(* IEC 61131-3 sources: brOscatLib/oscatNetw (part 4) *)

(* ---- MB_CLIENT.st ---- *)
FUNCTION_BLOCK MB_CLIENT
    (*http://www.oscat.de/images/OSCATBasic/oscat_basic333_en.pdf#page=112*)
    CASE state OF

    00: (* Warten auf DELAY-Time *)
    	ton_1(IN:=ENABLE,PT:=DELAY);

    	IF ton_1.Q OR DELAY = T#0s THEN
    		ton_1(IN:=FALSE);
    		state := 20;
    		ip_state := BYTE#1; (* Anmelden *)
    	END_IF

    20: (* Bei IP_Control anmelden *)
    	IF ip_state = BYTE#3 THEN
    		(* IP Datenverkehr einrichten *)
    		IP_C.C_PORT := WORD#0; (* Port von IP_CONTROL verwenden *)
    		IP_C.C_IP := DWORD#0; (* IP von IP_CONTROL verwenden *)
    		IP_C.C_MODE := BOOL_TO_BYTE(UDP); (* Mode: 0=TCP+ACTIVE+IP , 1=UDP+ACTIVE+IP *)
    		IP_C.TIME_RESET := TRUE; (* Zeitueberwachung rücksetzen *)
    		IP_C.C_ENABLE := TRUE; (* Verbindungsaufbau freigeben *)
    		IP_C.R_OBSERVE := TRUE; (* Empfangsueberwachung *)
    		ERROR := DWORD#00; (* letzten Fehler rücksetzen *)

    		CASE FC OF
    		(******************************************************************)
    		1..2: (* 0x01 Read Coil Status , 0x02 Read Input Status *)
    			IF R_POINTS <= 2000 THEN
    				w_tmp := INT_TO_WORD(R_ADDR);
    				S_BUF.BUFFER[08] := WORD_TO_BYTE(SHR(w_tmp,8));
    				S_BUF.BUFFER[09] := WORD_TO_BYTE(w_tmp);
    				w_tmp := INT_TO_WORD(R_POINTS);
    				S_BUF.BUFFER[10] := WORD_TO_BYTE(SHR(w_tmp,8));
    				S_BUF.BUFFER[11] := WORD_TO_BYTE(w_tmp);
    				S_BUF.SIZE := UINT#12;
    				response :=	WORD_TO_INT(SHR(INT_TO_WORD(R_POINTS + 7),3));
    				comp := 7;
    			ELSE
    				ERROR := DWORD#2; (* ILLEGAL DATA ADDRESS *)
    			END_IF
    		(******************************************************************)
    		3..4: (* 0x03 Read Holding Registers , 0x04 Read Input Registers *)
    			IF R_POINTS <= 125 THEN
    				w_tmp := INT_TO_WORD(R_ADDR);
    				S_BUF.BUFFER[08] := WORD_TO_BYTE(SHR(w_tmp,8));
    				S_BUF.BUFFER[09] := WORD_TO_BYTE(w_tmp);
    				w_tmp := INT_TO_WORD(R_POINTS);
    				S_BUF.BUFFER[10] := WORD_TO_BYTE(SHR(w_tmp,8));
    				S_BUF.BUFFER[11] := WORD_TO_BYTE(w_tmp);
    				S_BUF.SIZE := UINT#12;
    				response :=	WORD_TO_INT(SHL(w_tmp,1));
    				comp := 7;
    			ELSE
    				ERROR := DWORD#2; (* ILLEGAL DATA ADDRESS *)
    			END_IF
    		(******************************************************************)
    		5:	(* 0x05 Force Single Coil *)
    			IF W_DATA_ADR <= DATA_SIZE THEN
    				w_tmp := INT_TO_WORD(W_ADDR);
    				S_BUF.BUFFER[08] := WORD_TO_BYTE(SHR(w_tmp,8));
    				S_BUF.BUFFER[09] := WORD_TO_BYTE(w_tmp);
    				S_BUF.BUFFER[10] := SEL((DATA[W_DATA_ADR] AND SHL(WORD#1,W_DATA_BITPOS))>WORD#00,BYTE#16#00,BYTE#16#FF);
    				S_BUF.BUFFER[11] := BYTE#00;
    				S_BUF.SIZE := UINT#12;
    				response := 3;
    				comp := 11;
    			ELSE
    				ERROR := DWORD#2; (* ILLEGAL DATA ADDRESS *)
    			END_IF
    		(******************************************************************)
    		6:	(* 0x06 Preset Single Register *)
    			IF W_DATA_ADR <= DATA_SIZE THEN
    				w_tmp := INT_TO_WORD(W_ADDR);
    				S_BUF.BUFFER[08] := WORD_TO_BYTE(SHR(w_tmp,8));
    				S_BUF.BUFFER[09] := WORD_TO_BYTE(w_tmp);
    				w_tmp := DATA[W_DATA_ADR];
    				S_BUF.BUFFER[10] := WORD_TO_BYTE(SHR(w_tmp,8));
    				S_BUF.BUFFER[11] := WORD_TO_BYTE(w_tmp);
    				S_BUF.SIZE := UINT#12;
    				response := 3;
    				comp := 11;
    			ELSE
    				ERROR := DWORD#2; (* ILLEGAL DATA ADDRESS *)
    			END_IF
    		(******************************************************************)
    		15:	(* 0x0F Force Multiple Coils *)
    			IF (WORD_TO_INT(SHR(INT_TO_WORD(WORD_TO_INT(SHL(INT_TO_WORD(W_DATA_ADR),4)) + W_POINTS + W_DATA_BITPOS + 15),4)) <= DATA_SIZE) AND W_POINTS <= 1968 THEN
    				w_tmp := INT_TO_WORD(W_ADDR);
    				S_BUF.BUFFER[08] := WORD_TO_BYTE(SHR(w_tmp,8));
    				S_BUF.BUFFER[09] := WORD_TO_BYTE(w_tmp);
    				w_tmp := INT_TO_WORD(W_POINTS);
    				S_BUF.BUFFER[10] := WORD_TO_BYTE(SHR(w_tmp,8));
    				S_BUF.BUFFER[11] := WORD_TO_BYTE(w_tmp);
    				S_BUF.BUFFER[12] := WORD_TO_BYTE(SHR(INT_TO_WORD(W_POINTS + 7),3));

    				w_mask := SHL(WORD#1,W_DATA_BITPOS);
    				bit_pos := 0;
    				w_tmp := WORD#00;
    				idx1 := 12;
    				idx2 := W_DATA_ADR;
    				FOR i := 1 TO W_POINTS DO
    					w_tmp :=BIT_LOAD_W(w_tmp,(DATA[idx2] AND w_mask) > WORD#0,bit_pos);
    					bit_pos := bit_pos + 1;
    					IF bit_pos > 7 OR i=W_POINTS THEN
    						bit_pos := 0;
    						idx1 := idx1 + 1;
    						S_BUF.BUFFER[idx1] := WORD_TO_BYTE(w_tmp);
    						w_tmp := WORD#0;
    					END_IF
    					w_mask := ROL(w_mask,1);
    					IF w_mask = WORD#1 THEN
    						idx2 := idx2 +1;
    					END_IF
    				END_FOR
    				S_BUF.SIZE := INT_TO_UINT(idx1 + 1);
    				response := 3;
    				comp := 11;
    			ELSE
    				ERROR := DWORD#2; (* ILLEGAL DATA ADDRESS *)
    			END_IF
    		(******************************************************************)
    		16:	(* 0x10 Write Multiple Registers *)
    			IF W_DATA_ADR + W_POINTS <= DATA_SIZE AND W_POINTS <= 123 THEN
    				w_tmp := INT_TO_WORD(W_ADDR);
    				S_BUF.BUFFER[08] := WORD_TO_BYTE(SHR(w_tmp,8));
    				S_BUF.BUFFER[09] := WORD_TO_BYTE(w_tmp);
    				w_tmp := INT_TO_WORD(W_POINTS);
    				S_BUF.BUFFER[10] := WORD_TO_BYTE(SHR(w_tmp,8));
    				S_BUF.BUFFER[11] := WORD_TO_BYTE(w_tmp);
    				S_BUF.BUFFER[12] := SHL(S_BUF.BUFFER[11],1);

    				idx1 := 11;
    				count := W_DATA_ADR + W_POINTS - 1;
    				FOR i := W_DATA_ADR TO count DO
    					idx1 := idx1 + 2;
    					idx2 := idx1 + 1; (* zweiter index für pcworx notwendig ! *)
    					w_tmp := DATA[i];
    					S_BUF.BUFFER[idx1] := WORD_TO_BYTE(SHR(w_tmp,8));
    					S_BUF.BUFFER[idx2] := WORD_TO_BYTE(w_tmp);
    				END_FOR

    				S_BUF.SIZE := INT_TO_UINT(idx2 + 1);
    				response := 3;
    				comp := 11;
    			ELSE
    				ERROR := DWORD#2; (* ILLEGAL DATA ADDRESS *)
    			END_IF
    		(******************************************************************)
    		22:	(* 0x16 mask Write Register *)
    			IF W_DATA_ADR + 2 <= DATA_SIZE THEN
    				w_tmp := INT_TO_WORD(W_ADDR);
    				S_BUF.BUFFER[08] := WORD_TO_BYTE(SHR(w_tmp,8));
    				S_BUF.BUFFER[09] := WORD_TO_BYTE(w_tmp);
    				idx1 := W_DATA_ADR;
    				w_tmp := DATA[idx1];
    				S_BUF.BUFFER[10] := WORD_TO_BYTE(SHR(w_tmp,8));
    				S_BUF.BUFFER[11] := WORD_TO_BYTE(w_tmp);
    				idx1 := idx1 +1;
    				w_tmp := DATA[idx1];
    				S_BUF.BUFFER[12] := WORD_TO_BYTE(SHR(w_tmp,8));
    				S_BUF.BUFFER[13] := WORD_TO_BYTE(w_tmp);

    				S_BUF.SIZE := UINT#14;
    				response := 5;
    				comp := 13;
    			ELSE
    				ERROR := DWORD#2; (* ILLEGAL DATA ADDRESS *)
    			END_IF
    		(******************************************************************)
    		23:	(* 0x17 Read/Write Multible Registers *)
    			IF W_DATA_ADR + W_POINTS <= DATA_SIZE AND W_POINTS <= 121 AND R_POINTS <= 125 THEN
    				idx1 := 15;
    				count := W_DATA_ADR + W_POINTS - 1;
    				FOR i := W_DATA_ADR TO count DO
    					idx1 := idx1 + 2;
    					idx2 := idx1 + 1; (* zweiter index für pcworx notwendig ! *)
    					w_tmp := DATA[i];
    					S_BUF.BUFFER[idx1] := WORD_TO_BYTE(SHR(w_tmp,8));
    					S_BUF.BUFFER[idx2] := WORD_TO_BYTE(w_tmp);
    				END_FOR

    				(* WRITE *)
    				w_tmp := INT_TO_WORD(W_ADDR);
    				S_BUF.BUFFER[12] := WORD_TO_BYTE(SHR(w_tmp,8));
    				S_BUF.BUFFER[13] := WORD_TO_BYTE(w_tmp);
    				w_tmp := INT_TO_WORD(W_POINTS);
    				S_BUF.BUFFER[14] := WORD_TO_BYTE(SHR(w_tmp,8));
    				S_BUF.BUFFER[15] := WORD_TO_BYTE(w_tmp);
    				S_BUF.BUFFER[16] := SHL(S_BUF.BUFFER[15],1);

    				(* READ *)
    				w_tmp := INT_TO_WORD(R_ADDR);
    				S_BUF.BUFFER[08] := WORD_TO_BYTE(SHR(w_tmp,8));
    				S_BUF.BUFFER[09] := WORD_TO_BYTE(w_tmp);
    				w_tmp := INT_TO_WORD(R_POINTS);
    				S_BUF.BUFFER[10] := WORD_TO_BYTE(SHR(w_tmp,8));
    				S_BUF.BUFFER[11] := WORD_TO_BYTE(w_tmp);

    				S_BUF.SIZE := INT_TO_UINT(idx2 + 1);
    				response := WORD_TO_INT(SHL(w_tmp,1));
    				comp := 7;
    			ELSE
    				ERROR := DWORD#2; (* ILLEGAL DATA ADDRESS *)
    			END_IF
    		(******************************************************************)

    		ELSE
    			ERROR := DWORD#00000001; (* ILLEGAL FUNCTION *)
    		END_CASE

    		(* Daten senden *)
    		IF ERROR = DWORD#00 THEN
    			transaction_id := transaction_id + 1;
    			w_tmp := UINT_TO_WORD(S_BUF.SIZE - UINT#6);
    			(* ---- H E A D E R --------------------------------------------------------------- *)
    			S_BUF.BUFFER[0] := ip_id; (* TRANSACTION-ID HI-Byte *)
    			S_BUF.BUFFER[1] := INT_TO_BYTE(transaction_id); (* TRANSACTION-ID LO-Byte *)
    			S_BUF.BUFFER[2] := BYTE#00; (* PROTOKOLL-ID HI-Byte *)
    			S_BUF.BUFFER[3] := BYTE#00; (* PROTOKOLL-ID LO-Byte *)
    			S_BUF.BUFFER[4] := WORD_TO_BYTE(SHR(w_tmp,8)); (* Laenge HI-Byte *)
    			S_BUF.BUFFER[5] := WORD_TO_BYTE(w_tmp); (* Laenge LO-Byte *)
    			S_BUF.BUFFER[6] := UNIT_ID; (* UNIT *)
    			S_BUF.BUFFER[7] := INT_TO_BYTE(FC); (* FUNCTION-CODE *)
    			(*----- END OF HEADER --------------------------------------------------------------*)
    			R_BUF.SIZE := UINT#0; (* Empfangsbuffer löschen *)
    			state := 30; (* wait for response *)
    		ELSE
    			ip_state := BYTE#4; (* Abmelden *)
    			state := 00;
    		END_IF
    	END_IF

    30: (* response *)
    	IF IP_C.ERROR <> DWORD#00 THEN
    		ERROR := IP_C.ERROR;
    		ip_state := BYTE#4; (* Abmelden *)
    		state := 00;
    	ELSIF S_BUF.SIZE = UINT#0 AND R_BUF.SIZE > UINT#0 THEN
    		(* erwartete länge in sendebuffer nachträglich eintragen um vergleich zu ermöglichen *)
    		w_tmp := INT_TO_WORD(response + 3);
    		S_BUF.BUFFER[4] := WORD_TO_BYTE(SHR(w_tmp,8));
    		S_BUF.BUFFER[5] := WORD_TO_BYTE(w_tmp);

    		FOR i := 0 TO comp DO
    			IF S_BUF.BUFFER[i] <> R_BUF.BUFFER[i] THEN EXIT; END_IF
    		END_FOR

    		IF R_BUF.SIZE >= UINT#9 AND R_BUF.BUFFER[7] > BYTE#128 THEN  (* Bit 7 = ERROR Message *)
    			ERROR := BYTE_TO_DWORD(R_BUF.BUFFER[8]);
    			ip_state := BYTE#4; (* Abmelden *)
    			state := 00;
    		ELSIF R_BUF.SIZE = INT_TO_UINT(response + 9) AND i > comp THEN
    			mask := SHL(DWORD#1,FC);
    			(* READ_COILS, READ_INPUT_DISCRETES *)
    			IF (mask AND DWORD#2#00000000_00000000_00000000_00000110) > DWORD#0 THEN (* FC 1,2 *)
    				IF WORD_TO_INT(SHR(INT_TO_WORD(WORD_TO_INT(SHL(INT_TO_WORD(R_DATA_ADR),4)) + R_POINTS + R_DATA_BITPOS + 15),4)) <= DATA_SIZE THEN
    					b_mask := BYTE#1;
    					idx1 := 09;
    					idx2 := R_DATA_ADR;
    					bit_pos := R_DATA_BITPOS;
    					FOR i := 1 TO R_POINTS DO
    						DATA[idx2]:=BIT_LOAD_W(DATA[idx2],(R_BUF.BUFFER[idx1] AND b_mask) > BYTE#0,bit_pos);
    						bit_pos := bit_pos + 1;
    						IF bit_pos > 15 THEN
    							idx2 := idx2 + 1;
    							bit_pos := 0;
    						END_IF
    						b_mask := ROL(b_mask,1);
    						IF b_mask = BYTE#1 THEN
    							idx1 := idx1 + 1;
    						END_IF
    					END_FOR
    				ELSE
    					ERROR := DWORD#2; (* ILLEGAL DATA ADDRESS *)
    				END_IF

    			(* READ_MULTIPLE_REGISTERS, READ_INPUT_REGISTERS, READ_WRITE_REGISTERS *)
    			ELSIF (mask AND DWORD#2#00000000_10000000_00000000_00011000) > DWORD#0 THEN (* FC 3,4,23 *)
    				IF R_DATA_ADR + R_POINTS <= DATA_SIZE THEN
    					stop := R_DATA_ADR + R_POINTS -1 ;
    					idx1 := 07;
    					FOR i := R_DATA_ADR TO stop DO
    						idx1 := idx1 + 2;
    						idx2 := idx1 + 1;
    						DATA[i] := WORD_OF_BYTE(R_BUF.BUFFER[idx1],R_BUF.BUFFER[idx2]);
    					END_FOR
    				ELSE
    					ERROR := DWORD#2; (* ILLEGAL DATA ADDRESS *)
    				END_IF
    			ELSIF (mask AND DWORD#2#11111111_00111110_01111111_10000001) > DWORD#0 THEN (* ILLEGAL FUNCTION CODE ? *)
    				ERROR := DWORD#1; (* ILLEGAL FUNCTION *)
    			END_IF
    		ELSE
    			ERROR := DWORD#3; (* ILLEGAL DATA VALUE *)
    		END_IF

    		ip_state := BYTE#4; (* Abmelden *)
    		state := 00;
    		R_BUF.SIZE := UINT#0;

    	END_IF

    END_CASE

    (* ip_fifo *)
    ip_fifo(FIFO:=IP_C.FIFO,state:=ip_state,ID:=ip_id);
    BUSY := ip_state = BYTE#3;

    (* revision history
    ks	05. jan. 2009	rev 1.0
    	original version

    ks	28. jan. 2009	rev 1.1
    	network_buffer_short verwendet

    ks	20. oct. 2009	rev 1.2
    Networkbuffer und Buffer-funktionen auf Basis 0

    *)
END_FUNCTION_BLOCK

(* ---- MB_SERVER.st ---- *)
FUNCTION_BLOCK MB_SERVER
    (*http://www.oscat.de/images/OSCATBasic/oscat_basic333_en.pdf#page=116*)
    (* read system time *)
    tx := DWORD_TO_TIME(T_PLC_MS());

    FOR i := 1 TO 10 DO
    	IF VMAP[i].TIME_OUT > t#0s THEN
    		VMAP[i].TIME_OUT := VMAP[i].TIME_OUT + tx - last_cycle;
    	END_IF
    END_FOR
    last_cycle := tx;
    ip_error := IP_C.ERROR > DWORD#0;

    CASE state OF
    00: (* Warten auf Freigabe *)
    	IF ENABLE THEN
    		state := 10;
    		ip_state := BYTE#1; (* Anmelden *)
    	END_IF

    10: (* Bei IP_Control anmelden und auf freigabe warten *)
    	IF ip_state = BYTE#3 THEN

    		(* IP Datenverkehr einrichten *)
    		IP_C.C_PORT := WORD#0; (* Port von IP_CONTROL verwenden *)
    		IP_C.C_IP := DWORD#0; (* IP von IP_CONTROL verwenden *)
    		IP_C.C_MODE := SEL(UDP,BYTE#4,BYTE#5); (* Mode: 4=TCP+PASSIV+PORT , 5=UDP+PASSIV+PORT *)
    		IP_C.TIME_RESET := TRUE; (* Zeitueberwachung rücksetzen *)
    		IP_C.C_ENABLE := TRUE; (* Verbindungsaufbau freigeben *)
    		IP_C.R_OBSERVE := TRUE; (* keine Empfangsueberwachung *)
    		state := 20;
    	END_IF

    20:	IF NOT ip_error THEN
    		IF S_BUF.SIZE = UINT#0 AND R_BUF.SIZE > UINT#6 THEN	(* Datensenden nicht aktiv und Daten wurden empfangen *)
    			IF  R_BUF.SIZE = WORD_TO_UINT(WORD_OF_BYTE(R_BUF.BUFFER[4],R_BUF.BUFFER[5])) + UINT#6 THEN (* gültige Datenlänge *)
    				ERROR := DWORD#00; (* ERROR löschen *)

    				(* Header kopieren *)
    				FOR i := 0 TO 13 DO
    					S_BUF.BUFFER[i] := R_BUF.BUFFER[i];
    				END_FOR
    				fc := BYTE_TO_INT(R_BUF.BUFFER[7]);
    				adr1 := WORD_TO_INT(WORD_OF_BYTE(R_BUF.BUFFER[8],R_BUF.BUFFER[9]));
    				points := WORD_TO_INT(WORD_OF_BYTE(R_BUF.BUFFER[10],R_BUF.BUFFER[11]));

    				(* Virtual Address *)
    				MB_VMAP(VMAP:=VMAP,fc:=fc,V_ADR:=adr1,V_CNT:=points,SIZE:=DATA_SIZE);
    				adr1:=MB_VMAP.P_ADR;
    				bit_pos:=MB_VMAP.P_BIT;
    				ERROR:=BYTE_TO_DWORD(MB_VMAP.ERROR);

    				IF ERROR = DWORD#0 THEN
    					CASE fc OF
    					(*---------------------------------------------*)
    					1..2 : (* Read Coil Status / Read Input Status *)
    						count := 9; (* erstes Datenbyte *)
    						coils := BYTE#0;
    						mask := BYTE#1;
    						FOR i := 1 TO points DO
    							IF mask = BYTE#0 THEN
    								mask := BYTE#1;
    								S_BUF.BUFFER[count] := coils;
    								coils := BYTE#0;
    								count := count + 1;
    							END_IF
    							IF (DATA[adr1] AND SHL(WORD#1,bit_pos)) > WORD#0 THEN
    								coils := coils OR mask;
    							END_IF

    							bit_pos := bit_pos + 1;
    							IF bit_pos > 15 THEN
    								adr1 := adr1 + 1;
    								bit_pos := 0;
    							END_IF

    							mask := SHL(mask,1);
    						END_FOR
    						S_BUF.BUFFER[count] := coils;

    						S_BUF.BUFFER[8] := INT_TO_BYTE(count - 8); (* Bytecount *)
    						S_BUF.SIZE := INT_TO_UINT(count + 1);

    					(*--------------------------------------------------*)
    					3..4 : (* Read Holding Registers / Read Input Registers *)
    						idx1 := 07;
    						count := adr1 + points - 1;
    						FOR i := adr1 TO count DO
    							idx1 := idx1 + 2;
    							idx2 := idx1 + 1; (* zweiter index für pcworx notwendig ! *)
    							w_tmp := DATA[i];
    							S_BUF.BUFFER[idx1] := WORD_TO_BYTE(SHR(w_tmp,8));
    							S_BUF.BUFFER[idx2] := WORD_TO_BYTE(w_tmp);
    						END_FOR
    						S_BUF.BUFFER[8] := SHL(INT_TO_BYTE(points),1); (* Anzahl Register in Bytes *)
    						S_BUF.SIZE := INT_TO_UINT(idx2 + 1);
    					(*--------------------------------------------------*)
    					5 : (* Force Single Coil *)
    						DATA[adr1]:=BIT_LOAD_W(DATA[adr1],R_BUF.BUFFER[10] > BYTE#0,bit_pos);
    						S_BUF.SIZE := UINT#12;
    					(*--------------------------------------------------*)
    					6 : (* Preset Single Register *)
    						DATA[adr1] := WORD_OF_BYTE(R_BUF.BUFFER[10],R_BUF.BUFFER[11]);
    						S_BUF.SIZE := UINT#12;
    					(*--------------------------------------------------*)
    					15 : (* Force Multible coils *)
    						mask := BYTE#1;
    						idx1 := 13;
    						FOR i := 1 TO points DO
    							DATA[adr1]:=BIT_LOAD_W(DATA[adr1],(R_BUF.BUFFER[idx1] AND mask) > BYTE#0,bit_pos);
    							bit_pos := bit_pos + 1;
    							IF bit_pos > 15 THEN
    								adr1:= adr1 + 1;
    								bit_pos := 0;
    							END_IF
    							mask := ROL(mask,1);
    							IF mask = BYTE#1 THEN
    								idx1 := idx1 +1;
    							END_IF
    						END_FOR
    						S_BUF.SIZE := UINT#12;
    					(*--------------------------------------------------*)
    					16 : (* Preset Multiple Registers	*)
    						idx1 := 11;
    						count := adr1 + points - 1;
    						FOR i := adr1 TO count DO
    							idx1 := idx1 + 2;
    	 						idx2 := idx1 + 1;
    							DATA[i] := WORD_OF_BYTE(R_BUF.BUFFER[idx1],R_BUF.BUFFER[idx2]);
    						END_FOR
    						S_BUF.SIZE := UINT#12;
    					(*--------------------------------------------------*)
    					22 : (* mask Write Register *)
    						w_tmp := WORD_OF_BYTE(R_BUF.BUFFER[10],R_BUF.BUFFER[11]); (* and mask *)
    						DATA[adr1] := (DATA[adr1] AND w_tmp) OR (WORD_OF_BYTE(R_BUF.BUFFER[12],R_BUF.BUFFER[13]) AND (NOT w_tmp));
    						S_BUF.SIZE := UINT#14;
    					(*--------------------------------------------------*)
    					23 : (* Read / Write Registers	*)
    						(*--- Write-Register -----------------------------------*)
    						adr2 := WORD_TO_INT(WORD_OF_BYTE(R_BUF.BUFFER[12],R_BUF.BUFFER[13]));
    						points2 := WORD_TO_INT(WORD_OF_BYTE(R_BUF.BUFFER[14],R_BUF.BUFFER[15]));

    						(* Virtual Address Write Register *)
    						MB_VMAP(VMAP:=VMAP,fc:=16,V_ADR:=adr2,V_CNT:=points2,SIZE:=DATA_SIZE);
    						adr2:=MB_VMAP.P_ADR;
    						ERROR:=BYTE_TO_DWORD(MB_VMAP.ERROR);

    						IF ERROR = DWORD#0 THEN
    							idx1 := 15;
    							count := adr2 + points2 - 1;
    							FOR i := adr2 TO count DO
    								idx1 := idx1 + 2;
    	 							idx2 := idx1 + 1; (* zweiter index für pcworx notwendig ! *)
    								DATA[i] := WORD_OF_BYTE(R_BUF.BUFFER[idx1],R_BUF.BUFFER[idx2]);
    							END_FOR

    							(*--- Read-Register -----------------------------------*)
    							idx1 := 07;
    							count := adr1 + points - 1;
    							FOR i := adr1 TO count DO
    								idx1 := idx1 + 2;
    								idx2 := idx1 + 1; (* zweiter index für pcworx notwendig ! *)
    								w_tmp := DATA[i];
    								S_BUF.BUFFER[idx1] := WORD_TO_BYTE(SHR(w_tmp,8));
    								S_BUF.BUFFER[idx2] := WORD_TO_BYTE(w_tmp);
    							END_FOR
    							S_BUF.BUFFER[8] := SHL(INT_TO_BYTE(points),1); (* Anzahl Register in Bytes *)
    							S_BUF.SIZE := INT_TO_UINT(idx2 + 1);

    						END_IF

    					(*--------------------------------------------------*)
    					ELSE
    						ERROR := DWORD#01; (* ILLEGAL FUNCTION *)
    					END_CASE
    				END_IF
    			END_IF

    			IF ERROR > DWORD#0 THEN
    				S_BUF.BUFFER[7] := S_BUF.BUFFER[7] OR BYTE#2#1000_0000; (* Fehlerbit setzen *)
    				S_BUF.BUFFER[8] := DWORD_TO_BYTE(ERROR);
    				S_BUF.SIZE := UINT#9;
    			END_IF

    			S_BUF.BUFFER[4] := BYTE#0; (* high Byte *)
    			S_BUF.BUFFER[5] := UINT_TO_BYTE(S_BUF.SIZE - UINT#6); (* Längenfeld eintragen - nur low byte *)

    		END_IF
    	ELSE
    		ERROR := IP_C.ERROR;
    	END_IF

    	t(IN:= ip_error, PT:=t#2s);
    	IF t.Q THEN
    		IP_C.TIME_RESET := TRUE; (* ERROR Reset *)
    	END_IF

    	R_BUF.SIZE := UINT#0; (* Empfangsdaten zerstören *)

    	IF ENABLE = FALSE OR t.Q THEN
    	    ip_state := BYTE#4; (* Abmelden *)
    		state := 00;
    		IP_C.C_ENABLE := FALSE;
    	END_IF
    END_CASE

    (* IP_FIFO *)
    IP_FIFO(FIFO:=IP_C.FIFO,state:=ip_state,ID:=ip_id);

    (* revision history
    ks	05. jan. 2009	rev 1.0
    	original version

    ks	28. jan. 2009	rev 1.1
    	network_buffer_short verwendet

    ks	20. oct. 2009	rev 1.2
    	change lokal-var adr to adr1,Networkbuffer und Buffer-funktionen auf Basis 0

    ks	17. may. 2011	rev 1.3
    	automatischer re-connect

    ks	05. may. 2012	rev 1.4
    	timeoutüberwachung für re-connect
    *)
END_FUNCTION_BLOCK

(* ---- MB_SERVER_1.st ---- *)
FUNCTION_BLOCK MB_SERVER_1
    (*http://www.oscat.de/images/OSCATBasic/oscat_basic333_en.pdf#page=116*)
    (* read system time *)
    tx := DWORD_TO_TIME(T_PLC_MS());

    FOR i := 1 TO 10 DO
    	IF VMAP[i].TIME_OUT > t#0s THEN
    		VMAP[i].TIME_OUT := VMAP[i].TIME_OUT + tx - last_cycle;
    	END_IF
    END_FOR
    last_cycle := tx;
    ip_error := IP_C.ERROR > DWORD#0;

    CASE state OF
    00: (* Warten auf Freigabe *)
    	IF ENABLE THEN
    		state := 10;
    		ip_state := BYTE#1; (* Anmelden *)
    	END_IF

    10: (* Bei IP_Control anmelden und auf freigabe warten *)
    	IF ip_state = BYTE#3 THEN

    		(* IP Datenverkehr einrichten *)
    		IP_C.C_PORT := WORD#0; (* Port von IP_CONTROL verwenden *)
    		IP_C.C_IP := DWORD#0; (* IP von IP_CONTROL verwenden *)
    		IP_C.C_MODE := SEL(UDP,BYTE#4,BYTE#5); (* Mode: 4=TCP+PASSIV+PORT , 5=UDP+PASSIV+PORT *)
    		IP_C.TIME_RESET := TRUE; (* Zeitueberwachung rücksetzen *)
    		IP_C.C_ENABLE := TRUE; (* Verbindungsaufbau freigeben *)
    		IP_C.R_OBSERVE := FALSE; (* keine Empfangsueberwachung *)
    		state := 20;
    	END_IF

    20:	IF NOT ip_error THEN
    		IF S_BUF.SIZE = UINT#0 AND R_BUF.SIZE > UINT#6 THEN	(* Datensenden nicht aktiv und Daten wurden empfangen *)
    			IF  R_BUF.SIZE = WORD_TO_UINT(WORD_OF_BYTE(R_BUF.BUFFER[4],R_BUF.BUFFER[5])) + UINT#6 THEN (* gültige Datenlänge *)
    				ERROR := DWORD#00; (* ERROR löschen *)

    				(* Header kopieren *)
    				FOR i := 0 TO 13 DO
    					S_BUF.BUFFER[i] := R_BUF.BUFFER[i];
    				END_FOR
    				fc := BYTE_TO_INT(R_BUF.BUFFER[7]);
    				adr1 := WORD_TO_INT(WORD_OF_BYTE(R_BUF.BUFFER[8],R_BUF.BUFFER[9]));
    				points := WORD_TO_INT(WORD_OF_BYTE(R_BUF.BUFFER[10],R_BUF.BUFFER[11]));

    				(* Virtual Address *)
    				MB_VMAP(VMAP:=VMAP,fc:=fc,V_ADR:=adr1,V_CNT:=points,SIZE:=DATA_SIZE);
    				adr1:=MB_VMAP.P_ADR;
    				bit_pos:=MB_VMAP.P_BIT;
    				ERROR:=BYTE_TO_DWORD(MB_VMAP.ERROR);

    				IF ERROR = DWORD#0 THEN
    					CASE fc OF
    					(*---------------------------------------------*)
    					1..2 : (* Read Coil Status / Read Input Status *)
    						count := 9; (* erstes Datenbyte *)
    						coils := BYTE#0;
    						mask := BYTE#1;
    						FOR i := 1 TO points DO
    							IF mask = BYTE#0 THEN
    								mask := BYTE#1;
    								S_BUF.BUFFER[count] := coils;
    								coils := BYTE#0;
    								count := count + 1;
    							END_IF
    							IF (DATA[adr1] AND SHL(WORD#1,bit_pos)) > WORD#0 THEN
    								coils := coils OR mask;
    							END_IF

    							bit_pos := bit_pos + 1;
    							IF bit_pos > 15 THEN
    								adr1 := adr1 + 1;
    								bit_pos := 0;
    							END_IF

    							mask := SHL(mask,1);
    						END_FOR
    						S_BUF.BUFFER[count] := coils;

    						S_BUF.BUFFER[8] := INT_TO_BYTE(count - 8); (* Bytecount *)
    						S_BUF.SIZE := INT_TO_UINT(count + 1);

    					(*--------------------------------------------------*)
    					3..4 : (* Read Holding Registers / Read Input Registers *)
    						idx1 := 07;
    						count := adr1 + points - 1;
    						FOR i := adr1 TO count DO
    							idx1 := idx1 + 2;
    							idx2 := idx1 + 1; (* zweiter index für pcworx notwendig ! *)
    							w_tmp := DATA[i];
    							S_BUF.BUFFER[idx1] := WORD_TO_BYTE(SHR(w_tmp,8));
    							S_BUF.BUFFER[idx2] := WORD_TO_BYTE(w_tmp);
    						END_FOR
    						S_BUF.BUFFER[8] := SHL(INT_TO_BYTE(points),1); (* Anzahl Register in Bytes *)
    						S_BUF.SIZE := INT_TO_UINT(idx2 + 1);
    					(*--------------------------------------------------*)
    					5 : (* Force Single Coil *)
    						DATA[adr1]:=BIT_LOAD_W(DATA[adr1],R_BUF.BUFFER[10] > BYTE#0,bit_pos);
    						S_BUF.SIZE := UINT#12;
    					(*--------------------------------------------------*)
    					6 : (* Preset Single Register *)
    						DATA[adr1] := WORD_OF_BYTE(R_BUF.BUFFER[10],R_BUF.BUFFER[11]);
    						S_BUF.SIZE := UINT#12;
    					(*--------------------------------------------------*)
    					15 : (* Force Multible coils *)
    						mask := BYTE#1;
    						idx1 := 13;
    						FOR i := 1 TO points DO
    							DATA[adr1]:=BIT_LOAD_W(DATA[adr1],(R_BUF.BUFFER[idx1] AND mask) > BYTE#0,bit_pos);
    							bit_pos := bit_pos + 1;
    							IF bit_pos > 15 THEN
    								adr1:= adr1 + 1;
    								bit_pos := 0;
    							END_IF
    							mask := ROL(mask,1);
    							IF mask = BYTE#1 THEN
    								idx1 := idx1 +1;
    							END_IF
    						END_FOR
    						S_BUF.SIZE := UINT#12;
    					(*--------------------------------------------------*)
    					16 : (* Preset Multiple Registers	*)
    						idx1 := 11;
    						count := adr1 + points - 1;
    						FOR i := adr1 TO count DO
    							idx1 := idx1 + 2;
    	 						idx2 := idx1 + 1;
    							DATA[i] := WORD_OF_BYTE(R_BUF.BUFFER[idx1],R_BUF.BUFFER[idx2]);
    						END_FOR
    						S_BUF.SIZE := UINT#12;
    					(*--------------------------------------------------*)
    					22 : (* mask Write Register *)
    						w_tmp := WORD_OF_BYTE(R_BUF.BUFFER[10],R_BUF.BUFFER[11]); (* and mask *)
    						DATA[adr1] := (DATA[adr1] AND w_tmp) OR (WORD_OF_BYTE(R_BUF.BUFFER[12],R_BUF.BUFFER[13]) AND (NOT w_tmp));
    						S_BUF.SIZE := UINT#14;
    					(*--------------------------------------------------*)
    					23 : (* Read / Write Registers	*)
    						(*--- Write-Register -----------------------------------*)
    						adr2 := WORD_TO_INT(WORD_OF_BYTE(R_BUF.BUFFER[12],R_BUF.BUFFER[13]));
    						points2 := WORD_TO_INT(WORD_OF_BYTE(R_BUF.BUFFER[14],R_BUF.BUFFER[15]));

    						(* Virtual Address Write Register *)
    						MB_VMAP(VMAP:=VMAP,fc:=16,V_ADR:=adr2,V_CNT:=points2,SIZE:=DATA_SIZE);
    						adr2:=MB_VMAP.P_ADR;
    						ERROR:=BYTE_TO_DWORD(MB_VMAP.ERROR);

    						IF ERROR = DWORD#0 THEN
    							idx1 := 15;
    							count := adr2 + points2 - 1;
    							FOR i := adr2 TO count DO
    								idx1 := idx1 + 2;
    	 							idx2 := idx1 + 1; (* zweiter index für pcworx notwendig ! *)
    								DATA[i] := WORD_OF_BYTE(R_BUF.BUFFER[idx1],R_BUF.BUFFER[idx2]);
    							END_FOR

    							(*--- Read-Register -----------------------------------*)
    							idx1 := 07;
    							count := adr1 + points - 1;
    							FOR i := adr1 TO count DO
    								idx1 := idx1 + 2;
    								idx2 := idx1 + 1; (* zweiter index für pcworx notwendig ! *)
    								w_tmp := DATA[i];
    								S_BUF.BUFFER[idx1] := WORD_TO_BYTE(SHR(w_tmp,8));
    								S_BUF.BUFFER[idx2] := WORD_TO_BYTE(w_tmp);
    							END_FOR
    							S_BUF.BUFFER[8] := SHL(INT_TO_BYTE(points),1); (* Anzahl Register in Bytes *)
    							S_BUF.SIZE := INT_TO_UINT(idx2 + 1);

    						END_IF

    					(*--------------------------------------------------*)
    					ELSE
    						ERROR := DWORD#01; (* ILLEGAL FUNCTION *)
    					END_CASE
    				END_IF
    			END_IF

    			IF ERROR > DWORD#0 THEN
    				S_BUF.BUFFER[7] := S_BUF.BUFFER[7] OR BYTE#2#1000_0000; (* Fehlerbit setzen *)
    				S_BUF.BUFFER[8] := DWORD_TO_BYTE(ERROR);
    				S_BUF.SIZE := UINT#9;
    			END_IF

    			S_BUF.BUFFER[4] := BYTE#0; (* high Byte *)
    			S_BUF.BUFFER[5] := UINT_TO_BYTE(S_BUF.SIZE - UINT#6); (* Längenfeld eintragen - nur low byte *)

    		END_IF
    	ELSE
    		ERROR := IP_C.ERROR;
    	END_IF

    	t(IN:= ip_error, PT:=t#5s);
    	IF t.Q THEN
    		IP_C.TIME_RESET := TRUE; (* ERROR Reset *)
    	END_IF

    	R_BUF.SIZE := UINT#0; (* Empfangsdaten zerstören *)

    	IF ENABLE = FALSE THEN
    	    ip_state := BYTE#4; (* Abmelden *)
    		state := 00;
    	END_IF
    END_CASE

    (* IP_FIFO *)
    IP_FIFO(FIFO:=IP_C.FIFO,state:=ip_state,ID:=ip_id);

    (* revision history
    ks	05. jan. 2009	rev 1.0
    	original version

    ks	28. jan. 2009	rev 1.1
    	network_buffer_short verwendet

    ks	20. oct. 2009	rev 1.2
    	change lokal-var adr to adr1,Networkbuffer und Buffer-funktionen auf Basis 0

    ks	17. may. 2011	rev 1.3
    	automatischer re-connect
    *)
END_FUNCTION_BLOCK

(* ---- MB_VMAP.st ---- *)
FUNCTION_BLOCK MB_VMAP
    (*http://www.oscat.de/images/OSCATNetwork/oscat_netlib121_en.pdf#page=118*)
    IF init = FALSE THEN
    	init := TRUE;
    	IF VMAP[1].FC = DWORD#0 THEN
    		VMAP[1].FC := DWORD#16#FFFF_FFFF;
    		VMAP[1].V_ADR := 0;
    		VMAP[1].V_SIZE := 256;
    		VMAP[1].P_ADR := 0;
    	END_IF
    END_IF

    ERROR := BYTE#02; (* ILLEGAL DATA ADDRESS *)
    mask := SHL(DWORD#1,FC);

    IF (mask AND DWORD#2#00000000_01000000_00000000_01100000) <> DWORD#0 THEN (* FC 5,6,22 *)
    	V_CNT := 1;
    ELSIF V_CNT = 0 THEN
    	RETURN;
    END_IF

    FOR i := 1 TO 10 DO
    	vopt := VMAP[i].FC;
    	IF (vopt AND mask) <> DWORD#0 THEN
    		vadr := VMAP[i].V_ADR;
    		vsize := VMAP[i].V_SIZE;
    		padr := VMAP[i].P_ADR;

    		IF (mask AND DWORD#2#00000000_00000000_10000000_00100110) <> DWORD#0 THEN (* FC 1,2,5,15 für Bit-Access *)
    			i_tmp := WORD_TO_INT(SHR(INT_TO_WORD(V_ADR + V_CNT -1),4))+1;
    			IF i_tmp <= SIZE AND i_tmp <= vsize THEN
    				w_tmp := INT_TO_WORD(V_ADR);
    				P_ADR := WORD_TO_INT(SHR(w_tmp,4)) + padr;
    				P_BIT := WORD_TO_INT(w_tmp AND WORD#16#000F);
    				ERROR := BYTE#0;
    				EXIT;
    			END_IF
    		ELSIF (mask AND DWORD#2#00000000_11000001_00000000_01011000) <> DWORD#0 THEN (* FC 3,4,6,16,22,23 für Register-Access *)
    			IF V_ADR >= vadr AND V_ADR + V_CNT <= vadr + vsize THEN (* gültiger virtueller bereich *)
    				P_ADR := V_ADR - vadr + padr; (* reale Adresse berechnen *)
    				IF P_ADR + V_CNT <= SIZE THEN (* bereichsueberschreitung ? *)
    					ERROR := BYTE#0;
    					EXIT;
    				END_IF
    			END_IF
    		ELSE
    			ERROR := BYTE#01; (* ILLEGAL FUNCTION *)
    			RETURN;
    		END_IF
    	END_IF
    END_FOR

    IF ERROR = BYTE#0 THEN
    	IF (mask AND DWORD#2#00000000_11000001_10000000_01100000) <> DWORD#0 THEN (* FC 5,6,15,16,22,23 Schreib-zugriff *)
    		VMAP[i].TIME_OUT := T#1ms;
    	END_IF
    END_IF

    (* revision history
    ks	05. jan. 2009	rev 1.0
    	original version

    ks	20. oct. 2009	rev 1.1
    	fehlerkorrektur in bitmaske

    *)
END_FUNCTION_BLOCK

(* ---- MD5_CRAM_AUTH.st ---- *)
FUNCTION_BLOCK MD5_CRAM_AUTH
    (*http://www.oscat.de/images/OSCATBasic/oscat_basic333_en.pdf#page=78*)
    CASE step OF

    0:	IF RUN THEN
    		step := 5;
    		str_192 := B64_TS;
    		b64d_run := TRUE;
    	END_IF

    5: IF b64d_done THEN (* IPAD Zyklus *)
    		b64d_run := FALSE;
    		xpad := 16#36;
    		md5_str1 := PASSWORD;
    		md5_str2 := str_144;
    		size := 64 + LEN(md5_str2);
    		md5_mode := 1;
    		step := 10;
    	END_IF

    10: IF md5_mode = 3 THEN (* OPAD Zyklus *)
    		md5_first := md5; (* md5 array vom IPAD sichern *)
    		xpad := 16#5C;
    		size := 64 + 16;
    		md5_mode := 1;
    		step := 20;
    	END_IF

    20: IF md5_mode = 3 THEN
    		md5_mode := 0;
    		str_144 := CONCAT(USERNAME , ' ');
    		str_144 := CONCAT(str_144 , MD5_TO_STRH(md5));
    		b64e_run := TRUE;
    		step := 30;
    	END_IF

    30: IF b64e_done THEN
    		AUTH_KEY := str_192;
    		b64e_run := FALSE;
    		RUN := FALSE;
    		step := 0; (* alles beendet !! *)
    	END_IF

    END_CASE

    (* ----------- md5 -------------- *)
    CASE md5_mode OF

    1:	n2 := LEN(md5_str1) - 1;
    	pt := ADR(md5_str1);
    	FOR n1 := 0 TO n2 DO (* string in buf kopieren *)
    		buf[n1] := pt XOR xpad;
    		pt := pt + 1;
    	END_FOR
    	FOR n1 := n2 + 1 TO 63 DO (* mit ipad füllen *)
    		buf[n1] := xpad;
    	END_FOR

    2:	(* Data copy and Calc *)
    	IF size > 0 AND pos >= 64 THEN
    		IF step = 20 THEN
    			FOR n1 := 0 TO 15 DO
    				buf[n1] := md5_first[n1];
    			END_FOR
    		ELSE
    			n2 := LEN(md5_str2) - 1;
    			pt := ADR(md5_str2);
    			FOR n1 := 0 TO n2 DO (* string in buf kopieren *)
    				buf[n1] := pt;
    				pt := pt + 1;
    			END_FOR
    		END_IF
    	END_IF

    END_CASE

    IF md5_mode > 0 THEN
    	MD5_STREAM(size:=size, MODE:=md5_mode, buf:=buf, md5:=md5, pos=>pos);
    END_IF

    BASE64_DECODE_STR(RUN:=b64d_run, STR1:=str_192, STR2:=str_144, DONE=>b64d_done);
    BASE64_ENCODE_STR(RUN:=b64e_run, STR1:=str_144, STR2:=str_192, DONE=>b64e_done);

    (* revision history

    hm		10. mai. 2010	rev 1.0
    	original version
    *)
END_FUNCTION_BLOCK

(* ---- MD5_STR.st ---- *)
FUNCTION_BLOCK MD5_STR
    (*http://www.oscat.de/images/OSCATNetwork/oscat_netlib121_en.pdf#page=80*)
    CASE mode OF
    0:	(* Wait für Start *)
    	IF RUN AND NOT run_last THEN
    		DONE := FALSE;
    		mode := 1; (* Initialisierung *)
    		size := LEN(STR);
    	END_IF

    2:	(* Data copy and Calc *)
    	IF size > 0 THEN
    		_STRING_TO_BUFFER(STR:=MID(STR, UDINT_TO_INT(size), UDINT_TO_INT(pos) + 1), pos:=0, PT:=ADR(buf), size:=SIZEOF(buf));
    	END_IF

    3:	DONE := TRUE;
    	mode := 0; (* Stop *)

    END_CASE

    IF mode > 0 THEN
    	MD5_STREAM(size:=size, mode:=mode, buf:=buf, MD5:=MD5, pos=>pos);
    END_IF

    run_last := RUN;

    (* revision history

    ks	6. dec. 2009 rev 1.0
    	original version

    *)
END_FUNCTION_BLOCK

(* ---- MD5_STREAM.st ---- *)
FUNCTION_BLOCK MD5_STREAM
    (*http://www.oscat.de/images/OSCATNetwork/oscat_netlib121_en.pdf#page=80*)
    CASE MODE OF

    1:	(* Initialisierung der hash-Werte *)
    	hash[0] := DWORD#16#67452301;
    	hash[1] := DWORD#16#EFCDAB89;
    	hash[2] := DWORD#16#98BADCFE;
    	hash[3] := DWORD#16#10325476;

    	block := SHR(SIZE,6) + BOOL_TO_UDINT((UDINT_TO_BYTE(SIZE) AND 16#3F) > 55);
    	pad_1 := FALSE;
    	POS := 0;
    	end := SIZE;
    	SIZE := MIN(64,end);
    	MODE := 2;

    2:	(* Fuell-Bytes anhängen *)
    	FOR n := UDINT_TO_INT(SIZE) TO 63 DO
    		BUF[n] := 0;
    	END_FOR

    	IF SIZE < 64 AND NOT pad_1 THEN
    		BUF[SIZE] := 2#1000_0000;
    		pad_1 := TRUE;
    	END_IF

    	POS := POS + SIZE;
    	SIZE := MIN(64,end - POS);

    	n := 0;	(* Byte-Array in DWORD-Array umkopieren *)
    	FOR n1 := 0 TO 15 DO
    		x[n1] := DWORD_OF_BYTE(BUF[n+3],BUF[n+2],BUF[n+1],BUF[n]); (* Little Endian Format *)
    		n := n + 4;
    	END_FOR

    	IF block = 0 THEN (* am Ende des letzten Blocks die Datenlänge eintragen *)
    		x[14] := SHL(UDINT_TO_DWORD(end),3); (* Anzahl Datenbits im Little-Endian Format eintragen *)
    		MODE := 3;
    	ELSE
    		block := block - 1;
    	END_IF

    	a := hash[0];
    	b := hash[1];
    	c := hash[2];
    	d := hash[3];

    	a := MD5_AUX(1, a, b, c, d, x[00], 07, 16#D76AA478); (* 01 *)
    	d := MD5_AUX(1, d, a, b, c, x[01], 12, 16#E8C7B756); (* 02 *)
    	c := MD5_AUX(1, c, d, a, b, x[02], 17, 16#242070DB); (* 03 *)
    	b := MD5_AUX(1, b, c, d, a, x[03], 22, 16#C1BDCEEE); (* 04 *)
    	a := MD5_AUX(1, a, b, c, d, x[04], 07, 16#F57C0FAF); (* 05 *)
    	d := MD5_AUX(1, d, a, b, c, x[05], 12, 16#4787C62A); (* 06 *)
    	c := MD5_AUX(1, c, d, a, b, x[06], 17, 16#A8304613); (* 07 *)
    	b := MD5_AUX(1, b, c, d, a, x[07], 22, 16#FD469501); (* 08 *)
    	a := MD5_AUX(1, a, b, c, d, x[08], 07, 16#698098D8); (* 09 *)
    	d := MD5_AUX(1, d, a, b, c, x[09], 12, 16#8B44F7AF); (* 10 *)
    	c := MD5_AUX(1, c, d, a, b, x[10], 17, 16#FFFF5BB1); (* 11 *)
    	b := MD5_AUX(1, b, c, d, a, x[11], 22, 16#895CD7BE); (* 12 *)
    	a := MD5_AUX(1, a, b, c, d, x[12], 07, 16#6B901122); (* 13 *)
    	d := MD5_AUX(1, d, a, b, c, x[13], 12, 16#FD987193); (* 14 *)
    	c := MD5_AUX(1, c, d, a, b, x[14], 17, 16#A679438E); (* 15 *)
    	b := MD5_AUX(1, b, c, d, a, x[15], 22, 16#49B40821); (* 16 *)

    	a := MD5_AUX(2, a, b, c, d, x[01], 05, 16#F61E2562); (* 17 *)
    	d := MD5_AUX(2, d, a, b, c, x[06], 09, 16#C040B340); (* 18 *)
    	c := MD5_AUX(2, c, d, a, b, x[11], 14, 16#265E5A51); (* 19 *)
    	b := MD5_AUX(2, b, c, d, a, x[00], 20, 16#E9B6C7AA); (* 20 *)
    	a := MD5_AUX(2, a, b, c, d, x[05], 05, 16#D62F105D); (* 21 *)
    	d := MD5_AUX(2, d, a, b, c, x[10], 09, 16#02441453); (* 22 *)
    	c := MD5_AUX(2, c, d, a, b, x[15], 14, 16#D8A1E681); (* 23 *)
    	b := MD5_AUX(2, b, c, d, a, x[04], 20, 16#E7D3FBC8); (* 24 *)
    	a := MD5_AUX(2, a, b, c, d, x[09], 05, 16#21E1CDE6); (* 25 *)
    	d := MD5_AUX(2, d, a, b, c, x[14], 09, 16#C33707D6); (* 26 *)
    	c := MD5_AUX(2, c, d, a, b, x[03], 14, 16#F4D50D87); (* 27 *)
    	b := MD5_AUX(2, b, c, d, a, x[08], 20, 16#455A14ED); (* 28 *)
    	a := MD5_AUX(2, a, b, c, d, x[13], 05, 16#A9E3E905); (* 29 *)
    	d := MD5_AUX(2, d, a, b, c, x[02], 09, 16#FCEFA3F8); (* 30 *)
    	c := MD5_AUX(2, c, d, a, b, x[07], 14, 16#676F02D9); (* 31 *)
    	b := MD5_AUX(2, b, c, d, a, x[12], 20, 16#8D2A4C8A); (* 32 *)

    	a := MD5_AUX(3, a, b, c, d, x[05], 04, 16#FFFA3942); (* 33 *)
    	d := MD5_AUX(3, d, a, b, c, x[08], 11, 16#8771F681); (* 34 *)
    	c := MD5_AUX(3, c, d, a, b, x[11], 16, 16#6D9D6122); (* 35 *)
    	b := MD5_AUX(3, b, c, d, a, x[14], 23, 16#FDE5380C); (* 36 *)
    	a := MD5_AUX(3, a, b, c, d, x[01], 04, 16#A4BEEA44); (* 37 *)
    	d := MD5_AUX(3, d, a, b, c, x[04], 11, 16#4BDECFA9); (* 38 *)
    	c := MD5_AUX(3, c, d, a, b, x[07], 16, 16#F6BB4B60); (* 39 *)
    	b := MD5_AUX(3, b, c, d, a, x[10], 23, 16#BEBFBC70); (* 40 *)
    	a := MD5_AUX(3, a, b, c, d, x[13], 04, 16#289B7EC6); (* 41 *)
    	d := MD5_AUX(3, d, a, b, c, x[00], 11, 16#EAA127FA); (* 42 *)
    	c := MD5_AUX(3, c, d, a, b, x[03], 16, 16#D4EF3085); (* 43 *)
    	b := MD5_AUX(3, b, c, d, a, x[06], 23, 16#04881D05); (* 44 *)
    	a := MD5_AUX(3, a, b, c, d, x[09], 04, 16#D9D4D039); (* 45 *)
    	d := MD5_AUX(3, d, a, b, c, x[12], 11, 16#E6DB99E5); (* 46 *)
    	c := MD5_AUX(3, c, d, a, b, x[15], 16, 16#1FA27CF8); (* 47 *)
    	b := MD5_AUX(3, b, c, d, a, x[02], 23, 16#C4AC5665); (* 48 *)

    	a := MD5_AUX(4, a, b, c, d, x[00], 06, 16#F4292244); (* 49 *)
    	d := MD5_AUX(4, d, a, b, c, x[07], 10, 16#432AFF97); (* 50 *)
    	c := MD5_AUX(4, c, d, a, b, x[14], 15, 16#AB9423A7); (* 51 *)
    	b := MD5_AUX(4, b, c, d, a, x[05], 21, 16#FC93A039); (* 52 *)
    	a := MD5_AUX(4, a, b, c, d, x[12], 06, 16#655B59C3); (* 53 *)
    	d := MD5_AUX(4, d, a, b, c, x[03], 10, 16#8F0CCC92); (* 54 *)
    	c := MD5_AUX(4, c, d, a, b, x[10], 15, 16#FFEFF47D); (* 55 *)
    	b := MD5_AUX(4, b, c, d, a, x[01], 21, 16#85845DD1); (* 56 *)
    	a := MD5_AUX(4, a, b, c, d, x[08], 06, 16#6FA87E4F); (* 57 *)
    	d := MD5_AUX(4, d, a, b, c, x[15], 10, 16#FE2CE6E0); (* 58 *)
    	c := MD5_AUX(4, c, d, a, b, x[06], 15, 16#A3014314); (* 59 *)
    	b := MD5_AUX(4, b, c, d, a, x[13], 21, 16#4E0811A1); (* 60 *)
    	a := MD5_AUX(4, a, b, c, d, x[04], 06, 16#F7537E82); (* 61 *)
    	d := MD5_AUX(4, d, a, b, c, x[11], 10, 16#BD3AF235); (* 62 *)
    	c := MD5_AUX(4, c, d, a, b, x[02], 15, 16#2AD7D2BB); (* 63 *)
    	b := MD5_AUX(4, b, c, d, a, x[09], 21, 16#EB86D391); (* 64 *)

    	hash[0] := hash[0] + a;
    	hash[1] := hash[1] + b;
    	hash[2] := hash[2] + c;
    	hash[3] := hash[3] + d;

    END_CASE

    IF MODE = 3 THEN
    	z := 0;
    	FOR n := 0 TO 3 DO (* von Little-Endian auf Big-Endian format konvertieren und DWORD auf BYTE-Array *)
    		FOR n1 := 0 TO 3 DO
    			MD5[z] := DWORD_TO_BYTE(hash[n]);
    			hash[n] := ROR(hash[n],8);
    			z := z + 1;
    		END_FOR
    	END_FOR
    END_IF

    (* revision history

    ks	6. dec. 2009 rev 1.0
    	original version

    *)
END_FUNCTION_BLOCK

(* ---- MOON_PHASE.st ---- *)
FUNCTION_BLOCK MOON_PHASE
    (*http://www.oscat.de/images/OSCATNetwork/oscat_netlib121_en.pdf#page=206*)
    IF XDT - last_dt > UPDATE THEN
    	x := (DT_TO_UDINT(XDT) - 603240) MOD 2551392;
    	PHASE := UDINT_TO_BYTE(SCALE * x / 2551392) ;
    	last_dt := XDT;
    END_IF

    (* revision history
    ks	15.may. 2011	rev 1.0
    	original version

    *)
END_FUNCTION_BLOCK

(* ---- MYSQL_AUTH.st ---- *)
FUNCTION_BLOCK MYSQL_AUTH
    (*http://www.oscat.de/images/OSCATBasic/oscat_basic333_en.pdf#page=1*)
    IF NOT RUN THEN RETURN; END_IF
    CASE step OF

    0:	CASE sha_mode OF
    	0:	sha_mode := 1; (* Initialisierung *)
    		size := INT_TO_UDINT(LEN(PASSWORD));
    		i2 := UDINT_TO_INT(size) - 1;
    		FOR i := 0 TO 63 DO
    			IF i <= i2 THEN
    				buf[i] := CODE(STR:=PASSWORD,pos:=i+1);
    			ELSE
    				buf[i] := BYTE#0;
    			END_IF
    		END_FOR

    	3:	scramble1 := SCRAMBLE;
    		sha_mode := 1; (* Initialisierung *)
    		size := UDINT#20;
    		FOR i := 0 TO 19 DO
    			buf[i] := scramble1[i];
    		END_FOR
    		step := 10;
    	END_CASE

    10:	IF sha_mode = 3 THEN
    		sha_mode := 1; (* Initialisierung *)
    		scramble2 := SCRAMBLE;
    		size := UDINT#40;
    		FOR i := 0 TO 19 DO
    			buf[i] := MESSAGE[i];
    			buf[i+20] := scramble2[i];
    		END_FOR
    		step :=20;
    	END_IF

    20:	IF sha_mode = 3 THEN
    		sha_mode := 0; (* Stop *)
    		FOR i:= 0 TO 19 DO
    			SCRAMBLE[i] := SCRAMBLE[i] XOR scramble1[i];
    		END_FOR
    		step :=0;
    		RUN := FALSE;
    	END_IF
    END_CASE

    SHA1_STREAM(size:=size, MODE:=sha_mode, buf:=buf, SHA1:=SCRAMBLE, pos=>pos);

    (* revision history
    ks	20. apr. 2012	rev 1.0
    	original version

    *)
END_FUNCTION_BLOCK

(* ---- MYSQL_CONTROL.st ---- *)
FUNCTION_BLOCK MYSQL_CONTROL
    (*http://www.oscat.de/images/OSCATBasic/oscat_basic333_en.pdf#page=1*)
    CASE step OF

    00:	IF COM.SQL_CON THEN
    		timeout1 := MAX(T#10s,COM.TIMEOUT);
    		timeout2 := timeout1 + T#1s;
    		INFO.SQL_ERROR := '';
    		COM.ERROR_C := DWORD#0;
    		COM.ERROR_T := BYTE#0;
    		URL_DATA := STRING_TO_URL(STR:=COM.SQL_URL,DEFAULT_PROTOCOL:='',DEFAULT_PATH:='/');
    		step := 10;
    	END_IF

    10:	IF DNS_CLIENT.DONE THEN
    		step := 20;
    	ELSIF DNS_CLIENT.ERROR <> DWORD#0 THEN
    		COM.ERROR_C := DNS_CLIENT.ERROR;
    		COM.ERROR_T := BYTE#1;
    		step := 980;
    	END_IF

    20:	(* MySQL Steuerkanal einrichten *)
    	IF URL_DATA.PORT = WORD#0 THEN
    		URL_DATA.PORT := WORD#3306; (* Standard Port *)
    	END_IF
    	IP_C.C_PORT := URL_DATA.PORT; (* Portnummer eintragen *)
      	IP_C.C_IP := DNS_CLIENT.IP4; (* IP eintragen *)
      	IP_C.C_MODE := BYTE#0; (* Mode: TCP+ACTIV+PORT *)
      	IP_C.TIME_RESET := TRUE; (* Zeitueberwachung rücksetzen *)
      	IP_C.C_ENABLE := TRUE; (* Verbindungsaufbau freigeben *)
      	IP_C.R_OBSERVE := TRUE; (* Empfangsueberwachung *)
    	COM.R_BUF.SIZE := UINT#0;
    	COM.SQL_RCV_STATE := BYTE#0;
    	step := 30;

    30:	IF COM.SQL_RCV_STATE = BYTE#1 THEN
    		INFO.SERVER_PROTOCOL_VERSION := COM.R_BUF.BUFFER[4];

    		(* ende markierung von string server_version suchen *)
    		idx2 := UINT_TO_INT(COM.R_BUF.SIZE) - 1;
    		FOR idx1 := 5 TO idx2 DO
    			IF COM.R_BUF.BUFFER[idx1] = BYTE#0 THEN EXIT; END_IF
    		END_FOR
    		idx1 := idx1 + 5; (* terminierung und thread-id überspringen *)

    		FOR idx2:=0 TO 7 DO	(* Byte 0-7 *)
    			scramble1_buffer[idx2] := COM.R_BUF.BUFFER[idx1];
    			idx1 := idx1 + 1;
    		END_FOR
    		idx1 := idx1 + 1;
    		idx2 := idx1 + 1;
    		INFO.SERVER_CAPABILITIES := WORD_OF_BYTE(COM.R_BUF.BUFFER[idx2], COM.R_BUF.BUFFER[idx1]);
    		idx1 := idx1 + 2;
    		INFO.SERVER_LANGUAGE := COM.R_BUF.BUFFER[idx1];
    		idx1 := idx1 + 1;
    		idx2 := idx1 + 1;
    		INFO.SERVER_STATUS := WORD_OF_BYTE(COM.R_BUF.BUFFER[idx2], COM.R_BUF.BUFFER[idx1]);
    		idx1 := idx1 + 15;

    		FOR idx2:=8 TO 19 DO	(* Byte 8-19 *)
    			scramble1_buffer[idx2] := COM.R_BUF.BUFFER[idx1];
    			idx1 := idx1 + 1;
    		END_FOR

    		IF INFO.SERVER_PROTOCOL_VERSION < BYTE#10 THEN  (* Error: protocol version zu niedrig *)
    			COM.ERROR_T := BYTE#2;
    			COM.ERROR_C := DWORD#1;
    			step := 980;
    		ELSIF URL_DATA.PASSWORD = '' THEN
    			step := 50;
    		ELSE
    			auth_password := URL_DATA.PASSWORD;
    			auth_run := TRUE;
    			step := 40;
    		END_IF
    	END_IF

    40:	MYSQL_AUTH(RUN:= auth_run,PASSWORD:= auth_password ,MESSAGE:= scramble1_buffer,SCRAMBLE:= scramble2_buffer);
    	IF NOT auth_run THEN
    		step := 50;
    	END_IF

    50: (* Client Authentication Packet *)
    	(* Byte 0-3 werden später eingetragen *)
    	COM.S_BUF.BUFFER[04] := BYTE_OF_DWORD(client_flags, BYTE#0); (* client_flags *)
    	COM.S_BUF.BUFFER[05] := BYTE_OF_DWORD(client_flags, BYTE#1);
    	COM.S_BUF.BUFFER[06] := BYTE_OF_DWORD(client_flags, BYTE#2);
    	COM.S_BUF.BUFFER[07] := BYTE_OF_DWORD(client_flags, BYTE#3);
    	COM.S_BUF.BUFFER[08] := BYTE_OF_DWORD(max_packet_size, BYTE#0); (* max_packet_size *)
    	COM.S_BUF.BUFFER[09] := BYTE_OF_DWORD(max_packet_size, BYTE#1);
    	COM.S_BUF.BUFFER[10] := BYTE_OF_DWORD(max_packet_size, BYTE#2);
    	COM.S_BUF.BUFFER[11] := BYTE_OF_DWORD(max_packet_size, BYTE#3);
    	COM.S_BUF.BUFFER[12] := charset_number; (* charset_number *)
    	FOR idx1 := 13 TO 35 DO (* 23 bytes filler always 0x00.. *)
    		COM.S_BUF.BUFFER[idx1] := BYTE#0;
    	END_FOR
    	idx3 := LEN(URL_DATA.USER);
    	FOR idx2 :=1 TO idx3 DO
    		COM.S_BUF.BUFFER[idx1] := CODE(URL_DATA.USER, idx2);
    		idx1 := idx1 + 1;
    	END_FOR
    	COM.S_BUF.BUFFER[idx1] := BYTE#0; (* String terminierung eintragen *)
    	idx1 := idx1 + 1;
    	IF LEN(URL_DATA.PASSWORD) = 0 THEN
    		COM.S_BUF.BUFFER[idx1] := BYTE#0; (* scramble_buff length *)
    	ELSE
    		COM.S_BUF.BUFFER[idx1] := BYTE#20; (* scramble_buff length *)
    		FOR idx2 :=0 TO 19 DO
    			idx1 := idx1 + 1;
    			COM.S_BUF.BUFFER[idx1] := scramble2_buffer[idx2];
    		END_FOR
    	END_IF
    	COM.S_BUF.SIZE  := INT_TO_UINT(idx1 + 1); (* Sendelänge eintragen *)

    	step := 60;

    60:	IF COM.SQL_RCV_STATE = BYTE#1 THEN
    		INFO.SQL_CONNECTED := TRUE;
    		step := 300;
    	END_IF

    (* ================================================== *)

    300:	step := SEL(COM.SQL_CON,700,310); (* Schritt-Selektion *)

    310:	step := 300; (* dummy step *)

    (* ================================================== *)

    700: (* COM_QUIT *)
    	COM.S_BUF.BUFFER[04] := BYTE#1; (* 0x01 COM_QUIT mysql_close *)
    	COM.S_BUF.SIZE := UINT#5; (* Sendelänge eintragen *)
    	COM.SQL_PACKET_NO := BYTE#255;
    	ip_c_red_disable := TRUE;
    	step := 710;

    710:	IF IP_C.C_STATE = BYTE#0 THEN (* Verbindung durch SQL-Server beendet ? *)
    		step := 980;
    	END_IF

    (* ================================================== *)

    980:IP_C.C_ENABLE := FALSE; (* MYSQL Steuerkanal schliessen *)
    	ip_c_red_disable := FALSE;
    	INFO.SQL_CONNECTED := FALSE;
    	COM.SQL_CON := FALSE;
    	COM.S_BUF.SIZE := UINT#0;
    	COM.R_BUF.SIZE := UINT#0;
    	snd_step := 0;
    	step := 990;
    	(*####################  DEBUG-MESSAGE  ###################################*)
    	(*IF _debug_enable THEN
    		LOG_CL.NEW_MSG := 'QUIT: ERROR CODE >~1< TYPE >~2<';
    		LOG_CL.PRINTF[1] := DWORD_TO_STRH(COM.ERROR_C);
    		LOG_CL.PRINTF[2] := BYTE_TO_STRING(COM.ERROR_T);
    		LOG_MSG();
    	END_IF*)
    	(*########################################################################*)

    990:IF IP_C.C_STATE = BYTE#0 THEN
    		step := 0;
    	END_IF

    END_CASE

    (* ++++++++++++++++++++++++++++++++++++++++++++++++++++++++++ *)

    IF step >= 30 THEN
    	IF COM.R_BUF.SIZE >= UINT#3 AND COM.SQL_RCV_STATE = BYTE#0 THEN (* Daten wurden empfangen ? *)
    		IF DWORD_TO_UINT(DWORD_OF_BYTE(BYTE#0, COM.R_BUF.BUFFER[2], COM.R_BUF.BUFFER[1], COM.R_BUF.BUFFER[0])) + UINT#4 = COM.R_BUF.SIZE THEN
    			COM.SQL_PACKET_NO := COM.R_BUF.BUFFER[3];
    			IF COM.R_BUF.BUFFER[4] = BYTE#16#FF THEN
    				idx2 := 13; (* Error String - Erstes Zeichen *)
    				idx3 := UINT_TO_INT(COM.R_BUF.SIZE) - 1; (* Error String - Letztes Zeichen *)
    				FOR idx1 := idx2 TO idx3 DO (* alle ' durch ´ ersetzen *)
    					IF COM.R_BUF.BUFFER[idx1] = BYTE#39 THEN
    						COM.R_BUF.BUFFER[idx1] := BYTE#96;
    					END_IF
    				END_FOR
    				INFO.SQL_ERROR := BUFFER_TO_STRING(PT:=ADR(COM.R_BUF.BUFFER),SIZE:=COM.R_BUF.SIZE,START:=INT_TO_UINT(idx2),STOP:=INT_TO_UINT(idx3));
    				COM.ERROR_T := BYTE#3;
    				COM.ERROR_C := DWORD_OF_BYTE(BYTE#0,BYTE#0,COM.R_BUF.BUFFER[6], COM.R_BUF.BUFFER[5]);
    				COM.SQL_RCV_STATE := BYTE#2;
    				COM.R_BUF.SIZE := UINT#0; (* Empfangsbuffer nach Fehler rücksetzen *)
    				step := 980;
    			ELSE
    				COM.SQL_RCV_STATE := BYTE#1;
    				IP_C.R_OBSERVE := FALSE;

    				(*####################  DEBUG-MESSAGE  ###################################*)
    				(*IF _debug_enable THEN
    					LOG_CL.NEW_MSG := 'RCV: size >~1<';
    					LOG_CL.PRINTF[1] := UINT_TO_STRING(COM.R_BUF.SIZE);
    					LOG_MSG();
    				END_IF*)
    				(*########################################################################*)
    			END_IF
    		END_IF
    	END_IF
    END_IF

    (* automatisches Datensenden *)

    CASE snd_step OF

    00:	IF step >= 20 AND COM.S_BUF.SIZE > UINT#0 THEN
    		dw_tmp := UINT_TO_DWORD(COM.S_BUF.SIZE - UINT#4); (* packet_length *)
    		COM.S_BUF.BUFFER[0] := BYTE_OF_DWORD(dw_tmp, BYTE#0);
    		COM.S_BUF.BUFFER[1] := BYTE_OF_DWORD(dw_tmp, BYTE#1);
    		COM.S_BUF.BUFFER[2] := 0;
    		COM.SQL_PACKET_NO := COM.SQL_PACKET_NO + 1;
    		COM.S_BUF.BUFFER[3] := COM.SQL_PACKET_NO;

    		IP_C.R_OBSERVE := TRUE;
    		COM.R_BUF.SIZE := UINT#0; (* Empfangsbuffer rücksetzen *)
    		COM.SQL_RCV_STATE := BYTE#0;

    	        (*####################  DEBUG-MESSAGE  ###################################*)
    	        (*IF _debug_enable THEN
    	          LOG_CL.NEW_MSG := 'SND: size >~1<';
    	          LOG_CL.PRINTF[1] := UINT_TO_STRING(COM.S_BUF.SIZE);
    	          LOG_MSG();
    	        END_IF*)
    	        (*########################################################################*)

    		snd_step := 10;
    	END_IF

    10:	IF COM.S_BUF.SIZE = UINT#0 THEN (* warten bis alle daten gesendet sind *)
    		snd_step := 0;
    	END_IF

    END_CASE

    (* Globale Fehlerbehandlung für Haupt-Routine *)
    IF COM.ERROR_T = BYTE#0 AND step > 20 THEN (* noch kein Fehler gespeichert und Hauptroutine aktiv *)
    	IF IP_C.ERROR > DWORD#0 AND IP_C.C_ENABLE AND NOT IP_C.TIME_RESET THEN  (* IP Control *)
    		IF ip_c_red_disable = FALSE OR IP_C.ERROR <> DWORD#16#FD000000 THEN
    			COM.ERROR_C := IP_C.ERROR;
    			COM.ERROR_T := BYTE#2;
    			step := 980;
    		END_IF
    	END_IF
    END_IF

    IF TON_WAIT.Q THEN (* Ablaufstörung - Schrittkette *)
    	COM.ERROR_C := INT_TO_DWORD(step); (* aktuellen Schritt eintragen *)
    	COM.ERROR_T := BYTE#5;
    	step := 980;
    END_IF

    (* ######################################################## *)

    DNS_CLIENT(IP_C:=IP_C, S_BUF:=COM.S_BUF, R_BUF:=COM.R_BUF, DOMAIN:=URL_DATA.DOMAIN, IP4_DNS:= COM.DNS_IP4, ACTIVATE:=step=10); (* DNS-Client *)
    IPC(IP:= DWORD#0, PORT:= WORD#0 , TIME_OUT:= timeout1, IP_C:= IP_C, S_BUF:= COM.S_BUF, R_BUF:= COM.R_BUF); (* MYSQL Steuerkanal *)

    TON_WAIT(IN:=step = last_step AND step > 0,PT:=timeout2);
    last_step := step;

    (* revision history
    ks	20. apr. 2012	rev 1.0
    	original version
    ks	14. oct. 2013	rev 1.1
    	DNS_CLIENT Fehler durch zugriffskonflikt zwischen DNS_CLIENT und mySQL auf S_BUF

    *)
END_FUNCTION_BLOCK

(* ---- NET_VAR_BOOL8.st ---- *)
FUNCTION_BLOCK NET_VAR_BOOL8
    (*http://www.oscat.de/images/OSCATNetwork/oscat_netlib121_en.pdf#page=200*)
    IF NOT init THEN
    	init := TRUE;
    	X.ID_MAX := X.ID_MAX + USINT#1;
    	ID := USINT_TO_BYTE(X.ID_MAX);
    END_IF

    IF X.STATE > BYTE#0 AND X.ERROR_ID = BYTE#0 THEN
    	index := X.index; (* PCWORX Workaround *)
    	IF INT_TO_UINT(index + 3) > X.BUF_SIZE THEN
    		X.ERROR_ID := ID;
    	ELSE
    		IF X.STATE = BYTE#1 THEN (* Daten schreiben *)
    			X.S_BUF.BUFFER[index] := ID; (* ID *)
    			index := index + 1;
    			X.S_BUF.BUFFER[index] := BYTE#4; (* TYPE BOOL8 *)
    			index := index + 1;
    			X.S_BUF.BUFFER[index] := BYTE_OF_BIT(IN1,IN2,IN3,IN4,IN5,IN6,IN7,IN8);
    			index := index + 1;

    		ELSIF X.STATE = BYTE#2 THEN (* Daten lesen *)
    			index2 := index + 1; (* PCWORX Workaround *)
    			IF X.R_BUF.BUFFER[index] <> ID OR X.R_BUF.BUFFER[index2] <> BYTE#4 THEN
    				X.ERROR_ID := ID;
    			ELSE
    				index := index + 2;
    				BYTE_TO_BITS(IN:=X.R_BUF.BUFFER[index]);
    				OUT1 := BYTE_TO_BITS.B0;
    				OUT2 := BYTE_TO_BITS.B1;
    				OUT3 := BYTE_TO_BITS.B2;
    				OUT4 := BYTE_TO_BITS.B3;
    				OUT5 := BYTE_TO_BITS.B4;
    				OUT6 := BYTE_TO_BITS.B5;
    				OUT7 := BYTE_TO_BITS.B6;
    				OUT8 := BYTE_TO_BITS.B7;
    				index := index + 1;
    			END_IF
    		END_IF
    		X.index := index;
    	END_IF
    END_IF

    (* revision history
    ks	15.may. 2011	rev 1.0
    	original version

    *)
END_FUNCTION_BLOCK

(* ---- NET_VAR_BUFFER.st ---- *)
FUNCTION_BLOCK NET_VAR_BUFFER
    (*http://www.oscat.de/images/OSCATNetwork/oscat_netlib121_en.pdf#page=201*)
    IF NOT init THEN
    	init := TRUE;
    	X.ID_MAX := X.ID_MAX + USINT#1;
    	ID := USINT_TO_BYTE(X.ID_MAX);
    END_IF

    IF X.STATE > BYTE#0 AND X.ERROR_ID = BYTE#0 THEN
    	index := X.index; (* PCWORX Workaround *)
    	IF X.STATE = BYTE#1 THEN (* Daten schreiben *)
    		size := SIZEOF(BUF_IN);
    		IF INT_TO_UINT(index + 3 + size) > X.BUF_SIZE THEN
    			X.ERROR_ID := ID;
    		ELSE
    			X.S_BUF.BUFFER[index] := ID; (* ID *)
    			index := index + 1;
    			X.S_BUF.BUFFER[index] := BYTE#20; (* TYPE BUFFER *)
    			index := index + 1;
    			X.S_BUF.BUFFER[index] := INT_TO_BYTE(size); (* Anzahl der Bytes *)
    				index := index + 1;
    			FOR index2 := 1 TO size DO
    				X.S_BUF.BUFFER[index] := BUF_IN[index2];
    				index := index + 1;
    			END_FOR
    		END_IF
    	ELSIF X.STATE = BYTE#2 THEN (* Daten lesen *)
    		index2 := index + 1; (* PCWORX Workaround *)
    		IF X.R_BUF.BUFFER[index] <> ID OR X.R_BUF.BUFFER[index2] <> BYTE#20 THEN
    			X.ERROR_ID := ID;
    		ELSE
    			index := index + 2;
    			size := BYTE_TO_INT(X.R_BUF.BUFFER[index]);
    			index := index + 1;
    			FOR index2 := 1 TO size DO
    				BUF_OUT[index2] := X.R_BUF.BUFFER[index];
    				index := index + 1;
    			END_FOR
    		END_IF
    	END_IF
    	X.index := index;
    END_IF

    (* revision history
    ks	15.may. 2011	rev 1.0
    	original version

    *)
END_FUNCTION_BLOCK

(* ---- NET_VAR_CONTROL.st ---- *)
FUNCTION_BLOCK NET_VAR_CONTROL
    (*http://www.oscat.de/images/OSCATNetwork/oscat_netlib121_en.pdf#page=199*)
    IF X.ERROR_ID > BYTE#0 THEN (* Schwere Fehler bei Variablenzuordnung vorhanden  !! *)
    	X.STATE := BYTE#0;
    	ERROR := BYTE_TO_DWORD(X.ERROR_ID);
    	X.ERROR_ID := BYTE#0;
    	step := 999;
    END_IF

    CASE step OF

    00:	IF ACTIVATE AND NOT activate_last OR reset THEN

            (*  TCP + MASTER = C_MODE 0 (TCP + ACTIVE + PORT + IP) *)
            (*  UDP + MASTER = C_MODE 1 (UDP + ACTIVE + PORT + IP) *)
            (*  TCP + SLAVE  = C_MODE 2 (TCP + PASSIV + PORT + IP) *)
            (*  UDP + SLAVE  = C_MODE 3 (UDP + PASSIV + PORT + IP) *)
    	IF MASTER THEN
    		IP_C.C_MODE := BYTE#0;
    		step := 100;
    	ELSE
    		IP_C.C_MODE := BYTE#2;
    		step := 200;
    	END_IF
            IF UDP THEN IP_C.C_MODE := IP_C.C_MODE OR BYTE#1; END_IF
    	  	IP_C.C_PORT := REMOTE_PORT; (* Portnummer eintragen *)
    	  	IP_C.C_IP := REMOTE_IP4; (* IP eintragen *)
    	  	IP_C.TIME_RESET := TRUE; (* Zeitueberwachung rücksetzen *)
    	  	IP_C.C_ENABLE := TRUE; (* Verbindungsaufbau freigeben *)
    	  	IP_C.R_OBSERVE := TRUE; (* Empfangsueberwachung *)
    		X.S_BUF.SIZE := UINT#0;
    		X.R_BUF.SIZE := UINT#0;
    		X.CYCLE := UDINT#0;
    		X.ERROR_ID := BYTE#0;
    		reset := FALSE;
    	END_IF

    (* ++++++++++++++++++++++++++++++++++++++++++++++ *)

    100:IF IP_C.C_STATE > BYTE#127 THEN (* Verbindung vorhanden *)
    		X.STATE := BYTE#1; (* Daten sammeln *)
    		X.BUF_SIZE := SIZEOF(X.S_BUF.BUFFER);
    		X.S_BUF.BUFFER[0] := UDINT_TO_BYTE(X.CYCLE);
    		X.INDEX := 1;
    		step := 110;
    	END_IF

    110:X.STATE := BYTE#0;
    	X.S_BUF.SIZE := INT_TO_UINT(X.INDEX); (* Datenlänge eintragen *)
    	step := 120;

    120:IF X.S_BUF.SIZE = UINT#0 AND X.R_BUF.SIZE >= UINT#1 THEN (* länge der empfangenen Daten prüfen *)
    		X.STATE := BYTE#2; (* Daten ausgeben *)
    		X.BUF_SIZE := X.R_BUF.SIZE;
    		X.INDEX := 1;
    		X.ERROR_ID := BYTE#0;
    		X.CYCLE := X.CYCLE + UDINT#1;
    		ERROR := DWORD#0; (* nach erfolgreichen Zyklus letzten Fehlercode löschen *)
    		RUN := TRUE;
    		step := 130;
    	END_IF

    130:X.STATE := BYTE#0;
    	X.R_BUF.SIZE := UINT#0;
    	IF NOT ACTIVATE THEN
    		step := 999; (* Beenden *)
    	ELSIF tscan.Q THEN
    		step := 100;
    	END_IF

    (* ++++++++++++++++++++++++++++++++++++++++++++++ *)

    200:IF X.R_BUF.SIZE >= UINT#1 THEN
    		X.STATE := BYTE#2; (* Daten ausgeben *)
    		X.BUF_SIZE := X.R_BUF.SIZE;
    		X.INDEX := 1;
    		step := 210;
    	END_IF

    210:X.STATE := BYTE#1; (* Daten sammeln *)
    	X.BUF_SIZE := SIZEOF(X.R_BUF.BUFFER);;
    	X.S_BUF.BUFFER[0] := X.R_BUF.BUFFER[0]; (* Cycle übernehmen *)
    	X.INDEX := 1;
    	X.R_BUF.SIZE := UINT#0;
    	step := 220;

    220:X.STATE := BYTE#0;
    	X.S_BUF.SIZE := INT_TO_UINT(X.INDEX); (* Datenlänge eintragen *)
    	step := 230;

    230:IF X.S_BUF.SIZE = UINT#0 THEN
    		ERROR := DWORD#0; (* nach erfolgreichen Zyklus letzten Fehlercode löschen *)
    		RUN := TRUE;
    		IF NOT ACTIVATE THEN
    			step := 999; (* Beenden *)
    		ELSE
    			step := 200;
    		END_IF
    	END_IF

    999:IP_C.C_ENABLE := FALSE; (* Beenden *)
    	RUN := FALSE;
    	step := 0;

    END_CASE

    (* ++++++++++++++++++++++++++++++++++++++++++++++ *)

    IPC(IP:= DWORD#0, PORT:= WORD#0 , TIME_OUT:= WATCHDOG, IP_C:= IP_C, S_BUF:= X.S_BUF, R_BUF:= X.R_BUF);

    IF IP_C.ERROR > DWORD#0 THEN
    	ERROR := IP_C.ERROR;
    	RUN := FALSE;
    	reset := TRUE;
    	step := 0;
    END_IF

    activate_last := ACTIVATE; (* letzten Status sichern zur Flankenerkennung *)
    tscan(IN:= step <> 110 ,PT:=SCAN_TIME);

    (* revision history
    ks	15.may. 2011	rev 1.0
    	original version

    *)
END_FUNCTION_BLOCK

(* ---- NET_VAR_DWORD8.st ---- *)
FUNCTION_BLOCK NET_VAR_DWORD8
    (*http://www.oscat.de/images/OSCATNetwork/oscat_netlib121_en.pdf#page=202*)
    IF NOT init THEN
    	init := TRUE;
    	X.ID_MAX := X.ID_MAX + USINT#1;
    	ID := USINT_TO_BYTE(X.ID_MAX);
    END_IF

    IF X.STATE > BYTE#0 AND X.ERROR_ID = BYTE#0 THEN
    	index := X.index; (* PCWORX Workaround *)
    	IF INT_TO_UINT(index + 34) > X.BUF_SIZE THEN  (* ID (1) + TYPE (1) + 8 X DWORD (4) *)
    		X.ERROR_ID := ID;
    	ELSE
    		IF X.STATE = BYTE#1 THEN (* Daten schreiben *)
    			ra[1] := IN1;
    			ra[2] := IN2;
    			ra[3] := IN3;
    			ra[4] := IN4;
    			ra[5] := IN5;
    			ra[6] := IN6;
    			ra[7] := IN7;
    			ra[8] := IN8;
    			X.S_BUF.BUFFER[index] := ID; (* ID *)
    			index := index + 1;
    			X.S_BUF.BUFFER[index] := BYTE#13; (* TYPE DWORD8 *)
    			index := index + 1;
    			FOR i2 := 1 TO 8 DO;
    				FOR i := 1 TO 4 DO;
    					X.S_BUF.BUFFER[index] := DWORD_TO_BYTE(ra[i2]);
    					ra[i2] := ROR(ra[i2],8);
    					index := index + 1;
    				END_FOR
    			END_FOR

    		ELSIF X.STATE = BYTE#2 THEN (* Daten lesen *)
    			index2 := index + 1; (* PCWORX Workaround *)
    			IF X.R_BUF.BUFFER[index] <> ID OR X.R_BUF.BUFFER[index2] <> BYTE#13 THEN (* TYPE DWORD8 *)
    				X.ERROR_ID := ID;
    			ELSE
    				index := index + 2;
    				FOR i2 := 1 TO 8 DO;
    					ra[i2] := DWORD#0;
    					FOR i := 1 TO 4 DO;
    						ra[i2] := ra[i2] OR BYTE_TO_DWORD(X.R_BUF.BUFFER[index]);
    						ra[i2] := ROR(ra[i2],8);
    						index := index + 1;
    					END_FOR
    				END_FOR
    				OUT1 := ra[1];
    				OUT2 := ra[2];
    				OUT3 := ra[3];
    				OUT4 := ra[4];
    				OUT5 := ra[5];
    				OUT6 := ra[6];
    				OUT7 := ra[7];
    				OUT8 := ra[8];
    			END_IF
    		END_IF
    		X.index := index;
    	END_IF
    END_IF

    (* revision history
    ks	15.may. 2011	rev 1.0
    	original version

    *)
END_FUNCTION_BLOCK

(* ---- NET_VAR_REAL8.st ---- *)
FUNCTION_BLOCK NET_VAR_REAL8
    (*http://www.oscat.de/images/OSCATNetwork/oscat_netlib121_en.pdf#page=202*)
    IF NOT init THEN
    	init := TRUE;
    	X.ID_MAX := X.ID_MAX + USINT#1;
    	ID := USINT_TO_BYTE(X.ID_MAX);
    END_IF

    IF X.STATE > BYTE#0 AND X.ERROR_ID = BYTE#0 THEN
    	index := X.index; (* PCWORX Workaround *)
    	IF INT_TO_UINT(index + 34) > X.BUF_SIZE THEN (* ID (1) + TYPE (1) + 8 X REAL (4) *)
    		X.ERROR_ID := ID;
    	ELSE
    		IF X.STATE = BYTE#1 THEN (* Daten schreiben *)
    			ra[1] := IN1;
    			ra[2] := IN2;
    			ra[3] := IN3;
    			ra[4] := IN4;
    			ra[5] := IN5;
    			ra[6] := IN6;
    			ra[7] := IN7;
    			ra[8] := IN8;
    			X.S_BUF.BUFFER[index] := ID; (* ID *)
    			index := index + 1;
    			X.S_BUF.BUFFER[index] := BYTE#15; (* TYPE REAL8 *)
    			index := index + 1;
    			FOR i2 := 1 TO 8 DO;
    				r_dw := REAL_TO_DW(X:=ra[i2]);
    				FOR i := 1 TO 4 DO;
    					X.S_BUF.BUFFER[index] := DWORD_TO_BYTE(r_dw);
    					r_dw := ROR(r_dw,8);
    					index := index + 1;
    				END_FOR
    			END_FOR

    		ELSIF X.STATE = BYTE#2 THEN (* Daten lesen *)
    			index2 := index + 1; (* PCWORX Workaround *)
    			IF X.R_BUF.BUFFER[index] <> ID OR X.R_BUF.BUFFER[index2] <> BYTE#15 THEN (* TYPE REAL8 *)
    				X.ERROR_ID := ID;
    			ELSE
    				index := index + 2;
    				FOR i2 := 1 TO 8 DO;
    					r_dw := DWORD#0;
    					FOR i := 1 TO 4 DO;
    						r_dw := r_dw OR BYTE_TO_DWORD(X.R_BUF.BUFFER[index]);
    						r_dw := ROR(r_dw,8);
    						index := index + 1;
    					END_FOR
    					ra[i2] := DW_TO_REAL(X:=r_dw);
    				END_FOR
    				OUT1 := ra[1];
    				OUT2 := ra[2];
    				OUT3 := ra[3];
    				OUT4 := ra[4];
    				OUT5 := ra[5];
    				OUT6 := ra[6];
    				OUT7 := ra[7];
    				OUT8 := ra[8];
    			END_IF
    		END_IF
    		X.index := index;
    	END_IF
    END_IF

    (* revision history
    ks	15.may. 2011	rev 1.0
    	original version

    *)
END_FUNCTION_BLOCK

(* ---- NET_VAR_STRING.st ---- *)
FUNCTION_BLOCK NET_VAR_STRING
    (*http://www.oscat.de/images/OSCATNetwork/oscat_netlib121_en.pdf#page=203*)
    IF NOT init THEN
    	init := TRUE;
    	X.ID_MAX := X.ID_MAX + USINT#1;
    	ID := USINT_TO_BYTE(X.ID_MAX);
    END_IF

    IF X.STATE > BYTE#0 AND X.ERROR_ID = BYTE#0 THEN
    	index := X.index; (* PCWORX Workaround *)
    	IF X.STATE = BYTE#1 THEN (* Daten schreiben *)
    		len_str := LEN(IN);
    		IF INT_TO_UINT(index + 3 + len_str) > X.BUF_SIZE THEN
    			X.ERROR_ID := ID;
    		ELSE
    			X.S_BUF.BUFFER[index] := ID; (* ID *)
    			index := index + 1;
    			X.S_BUF.BUFFER[index] := BYTE#6; (* TYPE REAL *)
    			index := index + 1;
    			X.S_BUF.BUFFER[index] := INT_TO_BYTE(len_str); (* Anzahl der Bytes *)
    			index := index + 1;
    			_STRING_TO_BUFFER(STR:=IN,POS:=index,PT:=ADR(X.S_BUF.BUFFER),SIZE:=X.BUF_SIZE);
    			index := index + len_str;
    		END_IF
    	ELSIF X.STATE = BYTE#2 THEN (* Daten lesen *)
    		index2 := index + 1; (* PCWORX Workaround *)
    		IF X.R_BUF.BUFFER[index] <> ID OR X.R_BUF.BUFFER[index2] <> BYTE#6 THEN
    			X.ERROR_ID := ID;
    		ELSE
    			index := index + 2;
    			len_str := BYTE_TO_INT(X.R_BUF.BUFFER[index]);
    			index2 := index + 1;
    			index := index2 + len_str;
    			IF len_str > 0 THEN
    				OUT := BUFFER_TO_STRING(PT:=ADR(X.R_BUF.BUFFER),SIZE:=X.BUF_SIZE,START:=INT_TO_UINT(index2),STOP:=INT_TO_UINT(index - 1));
    			ELSE
    				OUT := '';
    			END_IF
    		END_IF
    	END_IF
    	X.index := index;
    END_IF

    (* revision history
    ks	15.may. 2011	rev 1.0
    	original version

    *)
END_FUNCTION_BLOCK

(* ---- NET_VAR_X8.st ---- *)
FUNCTION_BLOCK NET_VAR_X8
    (*http://www.oscat.de/images/OSCATNetwork/oscat_netlib121_en.pdf#page=204*)
    IF NOT init THEN
    	init := TRUE;
    	X.ID_MAX := X.ID_MAX + USINT#1;
    	ID := USINT_TO_BYTE(X.ID_MAX);
    END_IF

    IF X.STATE > BYTE#0 AND X.ERROR_ID = BYTE#0 THEN
    	index := X.index; (* PCWORX Workaround *)
    	IF INT_TO_UINT(index + 34) > X.BUF_SIZE THEN  (* ID (1) + TYPE (1) + 8 X DWORD (4) *)
    		X.ERROR_ID := ID;
    	ELSE
    		IF X.STATE = BYTE#1 THEN (* Daten schreiben *)
    			ra[1] := REAL_TO_DW(X:=IN_REAL1);
    			ra[2] := REAL_TO_DW(X:=IN_REAL2);
    			ra[3] := DINT_TO_DWORD(IN_DINT1);
    			ra[4] := DINT_TO_DWORD(IN_DINT2);
    			ra[5] := UDINT_TO_DWORD(IN_UDINT1);
    			ra[6] := UDINT_TO_DWORD(IN_UDINT2);
    			ra[7] := IN_DWORD1;
    			ra[8] := IN_DWORD2;
    			X.S_BUF.BUFFER[index] := ID; (* ID *)
    			index := index + 1;
    			X.S_BUF.BUFFER[index] := BYTE#21; (* TYPE X8 *)
    			index := index + 1;
    			FOR i2 := 1 TO 8 DO;
    				FOR i := 1 TO 4 DO;
    					X.S_BUF.BUFFER[index] := DWORD_TO_BYTE(ra[i2]);
    					ra[i2] := ROR(ra[i2],8);
    					index := index + 1;
    				END_FOR
    			END_FOR

    		ELSIF X.STATE = BYTE#2 THEN (* Daten lesen *)
    			index2 := index + 1; (* PCWORX Workaround *)
    			IF X.R_BUF.BUFFER[index] <> ID OR X.R_BUF.BUFFER[index2] <> BYTE#21 THEN (* TYPE X8 *)
    				X.ERROR_ID := ID;
    			ELSE
    				index := index + 2;
    				FOR i2 := 1 TO 8 DO;
    					ra[i2] := DWORD#0;
    					FOR i := 1 TO 4 DO;
    						ra[i2] := ra[i2] OR BYTE_TO_DWORD(X.R_BUF.BUFFER[index]);
    						ra[i2] := ROR(ra[i2],8);
    						index := index + 1;
    					END_FOR
    				END_FOR
    				OUT_REAL1 := DW_TO_REAL(X:=ra[1]);
    				OUT_REAL2 := DW_TO_REAL(X:=ra[2]);
    				OUT_DINT1 := DWORD_TO_DINT(ra[3]);
    				OUT_DINT2 := DWORD_TO_DINT(ra[4]);
    				OUT_UDINT1 := DWORD_TO_UDINT(ra[5]);
    				OUT_UDINT2 := DWORD_TO_UDINT(ra[6]);
    				OUT_DWORD1 := ra[7];
    				OUT_DWORD2 := ra[8];
    			END_IF
    		END_IF
    		X.index := index;
    	END_IF
    END_IF

    (* revision history
    ks	15.may. 2011	rev 1.0
    	original version

    *)
END_FUNCTION_BLOCK
